(* Logix 5000 project; controller PLCbox vendor 1 type 14 code 149 rev 30.11; software revision 30.01; part 3 of 3 *)
(* tags used below, declared in another part *)
   HMI_BOOL : BOOL[32];
   PLC_BOOL : BOOL[32];
   System_REAL : REAL[10];
(* TestProgram, continued *)

ROUTINE _03_HMI   (* ladder *)
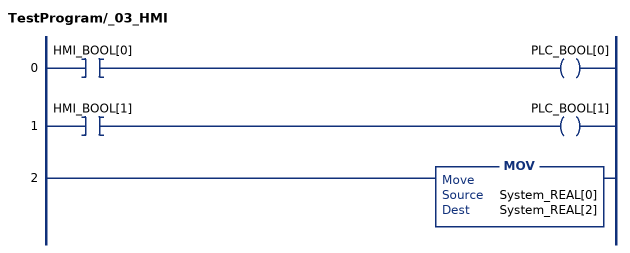
   0: XIC(HMI_BOOL[0])OTE(PLC_BOOL[0]);
   1: XIC(HMI_BOOL[1])OTE(PLC_BOOL[1]);
   2: MOV(System_REAL[0],System_REAL[2]);
END_ROUTINE

ROUTINE Main   (* ladder *)
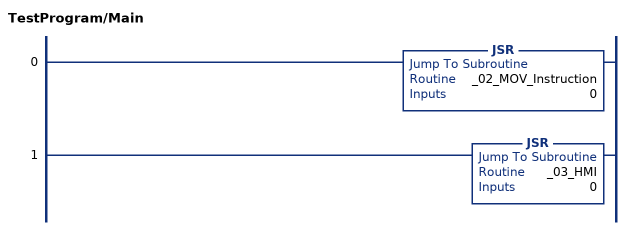
   0: JSR(_02_MOV_Instruction,0);
   1: JSR(_03_HMI,0);
END_ROUTINE
END_PROGRAM
